# EPICS substitutions: iocs/MC13/db/pmacStatus.substitutions
file "db/pmacStatus.db"
{
pattern
{SYS,            PMAC,    VERSION  PLC  PORT,  NAXES }
{"XF:06BM-CT",   "MC:13", "1"      5    "P0",  8     }
}
